{attribute 'GeneratedUsingTerminal: AT2040-0250-0021'}
{attribute addProperty BoxType "AT2040-0250-0021"}
{attribute addProperty Id "A_0108_AT2000_5233_0019_AT2000_5233AT2000_33A3DF1B80"}
{attribute addProperty CRC "193080036"}
{attribute addProperty Size "80"}
TYPE A_0036_AT2040_0250_0021_0B822AE4 EXTENDS AT2040_2EA6C9BF :
STRUCT
	{attribute addProperty Name "A_0108_AT2000_5233_0019_AT2000_5233"}
	{attribute addProperty PreviousPort "A_0036(AT2040-0250-0021) : B"}
	A_0108_AT2000_5233_0019_AT2000_5233 : AT2000_33A3DF1B;
END_STRUCT
END_TYPE

(* stored: Version 1.2.0.0, ProductVersion 3.1.4024.9
   DUT A_0036_AT2040_0250_0021_0B822AE4: Id {05dc0f3f-9436-4ba3-9448-cfd0c1f4dea8} *)
